TYPE ST_AlarmSirenHMI :
STRUCT
	sName		: STRING;	// Siren name
	nID			: INT;		// Alarm component ID
	bSiren		: BOOL;		// True if the siren is on
	bLight		: BOOL;		// True if the light is on
	bTamper		: BOOL;		// True if the siren is tampered with
END_STRUCT
END_TYPE

(* stored: Version 1.1.0.1, ProductVersion 3.1.4024.12
   DUT ST_AlarmSirenHMI: Id {bf9d0014-e1cc-44ce-b8d9-f8449be2fd73} *)
